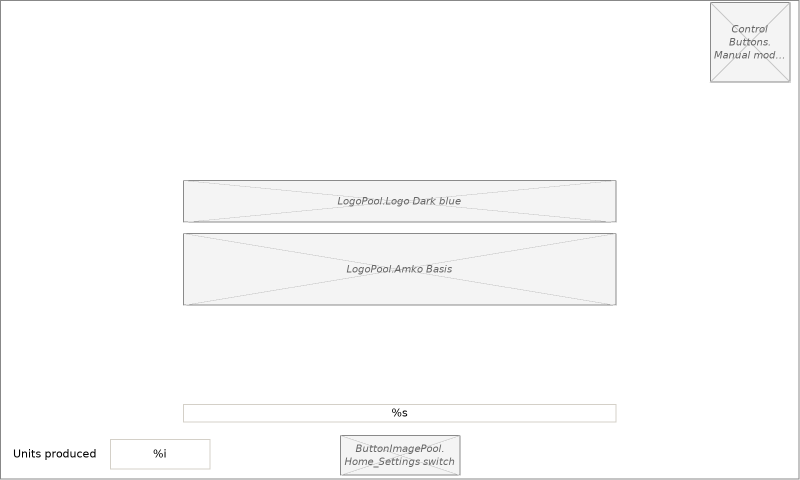
VISUALIZATION LogoScreen  // 800x480
    Rectangle (0,0 800x480)
    Image (183,180 433x42), image: LogoPool.Logo Dark blue
    Image (183,233 433x72), image: LogoPool.Amko Basis
    Textfield (183,404 433x18), "%s", tooltip "Operator messagages", text variable: GVL_Message.sOPeratorMessage
    Image (340,435 120x40), image: ButtonImagePool.Home_Settings switch
        OnMouseClick: execute { GVL_HMI.nStartVisu := E_BaseVisu.Parameter; }
    Image (710,2 80x80), image: ControlButtons.Manual mode Idle
        OnMouseClick: execute { GVL_HMI.nStartVisu := E_BaseVisu.Manual; }
    Textfield (110,439 100x30), "%i", text variable: GVL_Main.nTotalUnitsProduced
    Label (10,439 100x30), "Units produced"
END_VISUALIZATION

(* stored: Version 1.1.0.1, ProductVersion 3.1.4024.5
   Visu LogoScreen: Id {8e016bc8-ad21-4193-a4ea-5b7cd5d59e25} *)
